// TwinCAT 3 PLC project boor_tap_proces
// ProgramVersion: 3.1.4024.0
// libraries:
//   Tc2_Standard, * (Beckhoff Automation GmbH)
//   Tc2_System, * (Beckhoff Automation GmbH)
//   Tc3_Module, * (Beckhoff Automation GmbH)
//   VisuSymbols,3.5.10.0,System
// project tree:
//   / Boor_porces.TcPOU, Boren.TcTTO, GlobalTextList.TcGTLO, Hoofdschakelaar.TcTTO, Tappen.TcTTO, Visualization Manager.TcVMO (not stored)
//   GVLs/ GVL.TcGVL
//   POUs/ Hoofdschakelaar_.TcPOU, Tap_proces.TcPOU, MAIN.TcPOU
//   VISUs/ Visualization.TcVIS
// real-time tasks:
//   TASK PlcTask: cycle T#10ms, priority 20, ADS port 350
//   TASK Boren: cycle T#10ms, priority 21, ADS port 351
//   TASK Hoofdschakelaar: cycle T#10ms, priority 22, ADS port 352

CONFIGURATION boor_tap_proces
    RESOURCE PLC ON TwinCAT3
        TASK Boren(INTERVAL := T#10ms, PRIORITY := 21);
        TASK Hoofdschakelaar(INTERVAL := T#10ms, PRIORITY := 22);
        TASK Tappen(INTERVAL := T#10ms, PRIORITY := 20);
        PROGRAM Boor_porces WITH Boren : Boor_porces;
        PROGRAM Hoofdschakelaar_ WITH Hoofdschakelaar : Hoofdschakelaar_;
        PROGRAM Tap_proces WITH Tappen : Tap_proces;
    END_RESOURCE
END_CONFIGURATION

// ---- GVLs/GVL.TcGVL
{attribute 'qualified_only'}
VAR_GLOBAL
	
	
	//Hoofschakelaar
    Hoofdschakelaar: BOOL:= FALSE;       // Hoofdschakelaar (knop)
	Lamp_Hoofdschakelaar: BOOL:= FALSE;  //hoofdschakelaar aan (lamp)

	//Positie plaat
	Plaat_Gepositioneerd: BOOL := FALSE;   // Positie sensor plaat (knop/lamp)
	
    //boor proces
    Boor_Start: BOOL := FALSE;          //boor aan (lamp)
    Boor_Retour: BOOL := FALSE;         //Boor terug (lamp)
	Boor_aan: BOOL := FALSE;      		// Aanknop boor (knop)
	boor_Pos_Bereikt: BOOL := FALSE;    // Positie sensor boor onderin (sensor)
	boor_uit: BOOL := FALSE;			// uit knop boor (knop)
	
    //Tappen
	Tappen_Start: BOOL := FALSE;        //Tap aan (lamp)
    Tappen_Retour: BOOL := FALSE;       //Tap terug (lamp)
	Tappen_aan: BOOL := FALSE;      	// Aanknop Tap (knop)
	Tappen_Pos_Bereikt: BOOL := FALSE;  // Positie sensor Tap onderin (sensor)
	Tappen_uit: BOOL := FALSE;			// uit knop Tap (knop)
	
END_VAR

// ---- Boor_porces.TcPOU
PROGRAM Boor_porces
VAR
	Step: UINT:=0; 
END_VAR

CASE Step OF
	
	0: //Hoofdschakkelaar om zetten lamp gaat aan
	IF GVL.Hoofdschakelaar THEN
		Step := 1;
	END_IF
	
    1:  // Plaat in klem plaatsen sensor detecteerd of er een plaat in de klem zit
        IF GVL.Plaat_Gepositioneerd THEN
            Step := 2;
        END_IF

    2:  // Boor aan zetten 
        IF GVL.Boor_aan THEN
			GVL.Boor_Start := TRUE;
            Step := 3;
        END_IF
		
    3:  // Boor onderin, boor gaat terug naar boven
         IF GVL.boor_Pos_Bereikt THEN
            GVL.Boor_Retour := TRUE;
			GVL.Boor_Start := FALSE;
             Step := 4;
        END_IF

    4:  // Boor uitzetten
        IF GVL.Boor_uit THEN
            GVL.Boor_Retour := FALSE;
			Step:= 0;
        END_IF
		
END_CASE

END_PROGRAM

// ---- POUs/Hoofdschakelaar_.TcPOU
PROGRAM Hoofdschakelaar_
VAR
	 Step: UINT:=0; 
END_VAR


    // Hoofdschakelaar is true, turn on the lamp
   
        IF GVL.Hoofdschakelaar THEN
            GVL.Lamp_Hoofdschakelaar := TRUE;
		 ELSE
            GVL.Lamp_Hoofdschakelaar := FALSE;
        END_IF;

END_PROGRAM

// ---- POUs/Tap_proces.TcPOU
PROGRAM Tap_proces
VAR
	Step: UINT:=0; 
END_VAR

 CASE Step OF 
	
 	0: 
		IF GVL.Boor_uit AND GVL.Plaat_Gepositioneerd THEN
			Step :=1;
		END_IF

	1:  // Tappen aan zetten
        IF GVL.Tappen_aan THEN
			GVL.Tappen_Start := TRUE;
            Step := 2;
        END_IF
		
    2:  // Tap onderin, Tap gaat terug naar boven
         IF GVL.Tappen_Pos_Bereikt THEN
            GVL.Tappen_Retour := TRUE;
			GVL.Tappen_Start := FALSE;
             Step := 3;
        END_IF

    3:  // Tappen uitzetten
        IF GVL.Tappen_uit THEN
            GVL.Tappen_Retour := FALSE;
            Step := 4;
        END_IF
		
	4:   GVL.Plaat_Gepositioneerd := FALSE;
		 Step:= 1;		

END_CASE

END_PROGRAM

// ---- POUs/MAIN.TcPOU
PROGRAM MAIN
VAR
END_VAR

END_PROGRAM

// ---- GlobalTextList.TcGTLO
TEXTLIST GlobalTextList
  288 = 'Hoofdschakelaar'
  584 = 'Sensor plaat gepositioneerd'
END_TEXTLIST

// ---- VISUs/Visualization.TcVIS
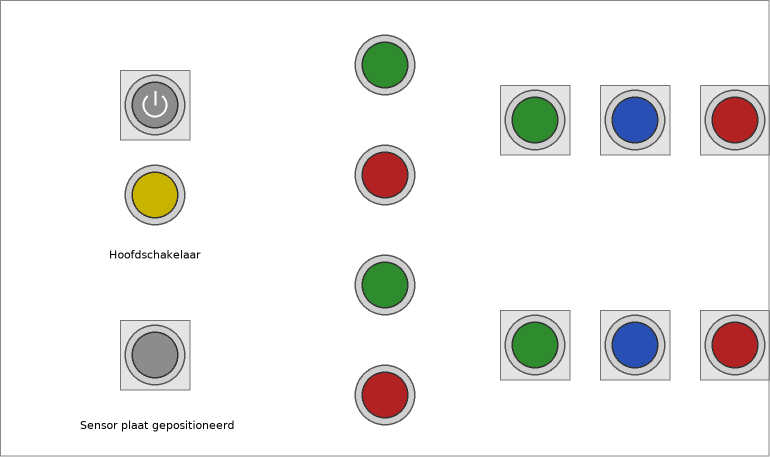
VISUALIZATION Visualization  // 770x457
    Lamp1 (350,30 70x70), variable: GVL.Boor_Start, style: Lamp-Lamp1-Green
    PowerSwitch (120,70 70x70), variable: GVL.Hoofdschakelaar, behaviour: TOGGLE, style: Switch-PowerSwitch-Gray
    Lamp1 (350,140 70x70), variable: GVL.Boor_Retour, style: Lamp-Lamp1-Red
    Lamp1 (350,250 70x70), variable: GVL.Tappen_Start, style: Lamp-Lamp1-Green
    PushSwitchLed (120,320 70x70), variable: GVL.Plaat_Gepositioneerd, behaviour: TOGGLE, style: Switch-PushSwitchLed-Gray
    Lamp1 (120,160 70x70), variable: GVL.Lamp_Hoofdschakelaar, style: Lamp-Lamp1-Yellow
    Label (80,240 150x30), "Hoofdschakelaar"
    Label (66,394 183x63), "Sensor plaat gepositioneerd"
    Lamp1 (350,360 70x70), variable: GVL.Tappen_Retour, style: Lamp-Lamp1-Red
    PushSwitch (500,85 70x70), variable: GVL.Boor_aan, behaviour: TAP, style: Switch-PushSwitch-Green
    PushSwitch (600,85 70x70), variable: GVL.boor_Pos_Bereikt, behaviour: TAP, style: Switch-PushSwitch-Blue
    PushSwitch (700,85 70x70), variable: GVL.boor_uit, behaviour: TAP, style: Switch-PushSwitch-Red
    PushSwitch (500,310 70x70), variable: GVL.Tappen_aan, behaviour: TAP, style: Switch-PushSwitch-Green
    PushSwitch (600,310 70x70), variable: GVL.Tappen_Pos_Bereikt, behaviour: TAP, style: Switch-PushSwitch-Blue
    PushSwitch (700,310 70x70), variable: GVL.Tappen_uit, behaviour: TAP, style: Switch-PushSwitch-Red
END_VISUALIZATION
